// TIA Portal V18 export
// export: Created 2026-06-08T16:08:49.7945797Z, ExportSetting WithDefaults, DisplayName Totally Integrated Automation Portal, DisplayVersion V18, DisplayName TIA Portal Openness, DisplayVersion V18, DisplayName TIA Portal Version Control Interface, DisplayVersion V18, DisplayName STEP 7 Professional, DisplayVersion V18, DisplayName STEP 7 Safety, DisplayVersion V18, DisplayName WinCC Professional, DisplayVersion V18
VAR_GLOBAL   // PLC tag table "TAG"
   Start AT %I0.0 : Bool;   // Nút nhấn Start
   Stop AT %I0.1 : Bool;   // Nút nhấn Stop
   Lamp AT %Q0.0 : Bool;   // Đèn hệ thống làm việc
   Sensor_Temperature AT %IW64 : Int;   // Cảm biến nhiệt độ
   QW_SSR AT %QW64 : Int;   // Đầu ra analog điều khiển SSR
   HMI_Start AT %M10.0 : Bool;   // Nút nhấn start trên Scada
   HMI_Stop AT %M10.1 : Bool;   // Nút nhấn Stop trên Scada
   HMI_Simulation AT %M10.2 : Bool;   // Nút mô phỏng tín hiệu nhiệt độ trên Scada
   HMI_Simu_Temperature AT %MW100 : Int;   // Mô phỏng nhiệt độ trên HMI
   HMI_Setting_Temperature AT %MD200 : Real;   // Cài đặt nhiệt độ cho máy sấy
   HMI_TT_Temperature AT %MD204 : Real;   // Nhiệt độ thực tế máy sấy
END_VAR
